FUNCTION TryConvert_LWORD_TO_SINT : BOOL
VAR_INPUT
	in : LWORD;
	out : REFERENCE TO SINT;
END_VAR

IF in > DatatypeLimits.MAX_VALUE_OF_LWORD_WHICH_CAN_BE_HELD_IN_A_SINT THEN
	RETURN;
END_IF

out := LWORD_TO_SINT(in);
TryConvert_LWORD_TO_SINT := TRUE;

END_FUNCTION

(* stored: Version 1.1.0.1, ProductVersion 3.1.4024.12
   POU TryConvert_LWORD_TO_SINT: Id {854885e5-e829-40a6-872b-3ff8da2067bd}, SpecialFunc None *)
